FUNCTION_BLOCK SEL_COLOR (* See SEL_ANY *)
  (* Standard: 61131-3 *)
  (* Version 0.0, 2004-12-15, JHC, Rockwell Automation, Converted from SRC format. *)
  (* Compiler header: package fb.rt.plc.select; *)
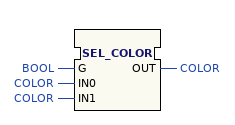
  VAR_INPUT
    G : BOOL;
    IN0 : COLOR;
    IN1 : COLOR;
  END_VAR
  VAR_OUTPUT
    OUT : COLOR;
  END_VAR
END_FUNCTION_BLOCK
